FUNCTION_BLOCK POU_ST_FUP
VAR_INPUT
END_VAR
VAR_OUTPUT
END_VAR
VAR
END_VAR

// NETWORK 1

END_FUNCTION_BLOCK

(* stored: Version 1.1.0.1, ProductVersion 3.1.4024.12
   POU POU_ST_FUP: Id {de978e52-b606-4a2c-a106-434353903a43}, SpecialFunc None *)
